(* Logix 5000 project; controller BoilerDemo vendor 1 type 14 code 164 rev 33.11; software revision 33.03 *)

TASK BoilerDemoTask (periodic, rate 75 ms, priority 10, watchdog 500 ms) : BoilerDemoProgram
TASK OvenDemoTask (continuous, watchdog 500 ms) : OvenDemo

MODULES
   Local : vendor 1 type 14 code 164 (ICP 1, rev 33.11)
END_MODULES

TYPE DATETIMESTRUCT :
STRUCT
   Year : DINT;
   Month : DINT;
   Day : DINT;
   Hour : DINT;
   Minute : DINT;
   Second : DINT;
   Microsecond : DINT;
END_STRUCT
END_TYPE

TYPE Motor :
STRUCT
   Power : REAL;
   Speed : INT;
   CmdOffOn : BOOL;
   SetSpeed : INT;
   Status : BOOL;
END_STRUCT
END_TYPE

TYPE Product :
STRUCT
   Product_id : INT;
   Product_name : STRING;
   Brand_id : INT;
   Category_id : INT;
   model_year : INT;
   list_price : REAL;
END_STRUCT
END_TYPE

TYPE Step :
STRUCT
   Num : INT;
   Time : TIMER;
   Step_Complete : BOOL;
   Prompt : BOOL;
   Prompt_Desc : STRING;
   Description : STRING;
END_STRUCT
END_TYPE

TYPE TankUDT :
STRUCT
   ValveInStatus : BOOL;
   ValveInCmd : BOOL;
   ValveOutStatus : BOOL;
   ValveOutCmd : BOOL;
   Level : REAL;
   SetPoint : REAL;
END_STRUCT
END_TYPE

ADD_ON_INSTRUCTION AOI_FaultGen   (* revision 1.2, vendor Rockwell Automation, ExecuteEnableInFalse *)
// Using random numbers [AOI_SIM_RNG_Simple] to generate 1-64 faults and their duration
// Revision note:
// Cfg_CycleTime changed to local tag (no need to have many configuration tags exposed)
// Help:
// This AOI uses Random Number ganerator to create up to 64 different outputus (BOOLs), each with different duration.
// ( Cfg_FaultOccurencesAll ) affects "probability" of TRUE value of all outputs ( F.x )
// ( Cfg_FaultOccurences[x] ) can be used to set the ratio among "probabilities" of individual outputs ( F.x ) getting true -> higher value, haigher probability
// Mechanism:
// - Value of the random number is between 0 and 1
// - Random number is generated every ( Cfg_CycleTime ) seconds
// - Value of Random numebr is checked, whether it falls in interval [0 - Cfg_FaultOccurenceAll]
// - If Random number is in the configured interval, then this interval is split into pieces:
//    where number of pieces to "split the interval into" is:
//    SUM of ( Cfg_FaultOccurences[] ) ... the count of Cfg_FaultOccurences members to use is ( Cfg_NumberOfFaults )
// - Each "output" (F.x) then has its "own" interval of the [0 - Cfg_FaultOccurenceAll]. If the Random number falls into the interval related to F.x, then F.x is set high
// - Reset of F.x to low is after a random time between ( Cfg_FaultDurationMin ) and ( Cfg_FaultDurationMax )
VAR_INPUT
   Cfg_NumberOfFaults : DINT := 1; {access None, visible}   // Number of faults to be generated (valid 1-64) value 0 resets the F (output) bits
   Cfg_FaultOccurenceAll : REAL := 0.05; {access None, visible}   // Probability of ANY fault occurence (valid 0-1)
   Cfg_FaultDurationMin : DINT := 15; {access None, visible}   // Minimum duration of fault [seconds]
   Cfg_FaultDurationMax : DINT := 75; {access None, visible}   // Maximum duration of fault [seconds]
END_VAR
VAR_OUTPUT
   F : LINT; {access None, visible}   // Generated fault bits
   RandomNr : REAL; {access Read Only, visible}
END_VAR
VAR
   TONs_FaultHold : TIMER[64]; {access None}
   z_CTRL : CONTROL := (LEN := 1); {access None}
   RandomNumber : REAL; {access None}
   TON_Cycle : TIMER := (PRE := 1500); {access None}
   Wrk_FaultOccurencesSUM : DINT; {access None}
   Wrk_Step : REAL; {access None}
   i : DINT; {access None}
   Wrk_StepLimit1 : REAL; {access None}
   Wrk_StepLimit2 : REAL; {access None}
   z_ONS : BOOL[64]; {access None}
   Random : AOI_SIM_RNG_Simple := (Seed := 521288629); {access None}
   Cfg_FaultOccurences : DINT[64] := ([0] := 100, [1] := 100, [2] := 100, [3] := 100, [4] := 100, [5] := 100, [6] := 100, [7] := 100, [8] := 100, [9] := 100, [10] := 100, [11] := 100, [12] := 100, [13] := 100, [14] := 100, [15] := 100, [16] := 100, [17] := 100, [18] := 100, [19] := 100, [20] := 100, [21] := 100, [22] := 100, [23] := 100, [24] := 100, [25] := 100, [26] := 100, [27] := 100, [28] := 100, [29] := 100, [30] := 100, [31] := 100, [32] := 100, [33] := 100, [34] := 100, [35] := 100, [36] := 100, [37] := 100, [38] := 100, [39] := 100, [40] := 100, [41] := 100, [42] := 100, [43] := 100, [44] := 100, [45] := 100, [46] := 100, [47] := 100, [48] := 100, [49] := 100, [50] := 100, [51] := 100, [52] := 100, [53] := 100, [54] := 100, [55] := 100, [56] := 100, [57] := 100, [58] := 100, [59] := 100,
        [60] := 100, [61] := 100, [62] := 100, [63] := 100);   // Each fault's "probability weight" (proportional to the other faults' "weights")
   i_max : DINT; {access None}
   Cfg_CycleTime : REAL := 1.5;   // Fault generation cycle time [seconds]
END_VAR

ROUTINE EnableInFalse   (* ladder *)
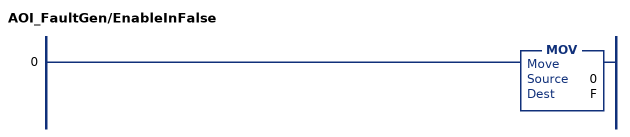
   0: MOV(0,F);
END_ROUTINE

ROUTINE Logic   (* ladder *)
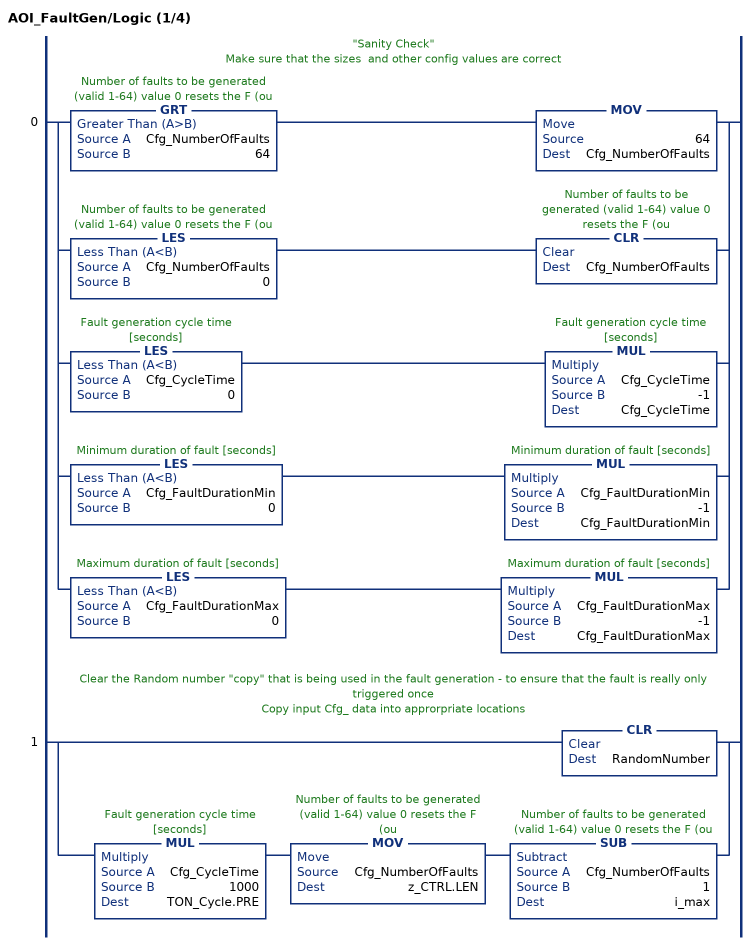
   // "Sanity Check"
   // Make sure that the sizes  and other config values are correct
   0: [GRT(Cfg_NumberOfFaults,64) MOV(64,Cfg_NumberOfFaults) ,LES(Cfg_NumberOfFaults,0) CLR(Cfg_NumberOfFaults) ,LES(Cfg_CycleTime,0) MUL(Cfg_CycleTime,-1,Cfg_CycleTime) ,LES(Cfg_FaultDurationMin,0) MUL(Cfg_FaultDurationMin,-1,Cfg_FaultDurationMin) ,LES(Cfg_FaultDurationMax,0) MUL(Cfg_FaultDurationMax,-1,Cfg_FaultDurationMax) ];
   // Clear the Random number "copy" that is being used in the fault generation - to ensure that the fault is really only triggered once
   // Copy input Cfg_ data into approrpriate locations
   1: [CLR(RandomNumber) ,MUL(Cfg_CycleTime,1000,TON_Cycle.PRE) MOV(Cfg_NumberOfFaults,z_CTRL.LEN) SUB(Cfg_NumberOfFaults,1,i_max) ];
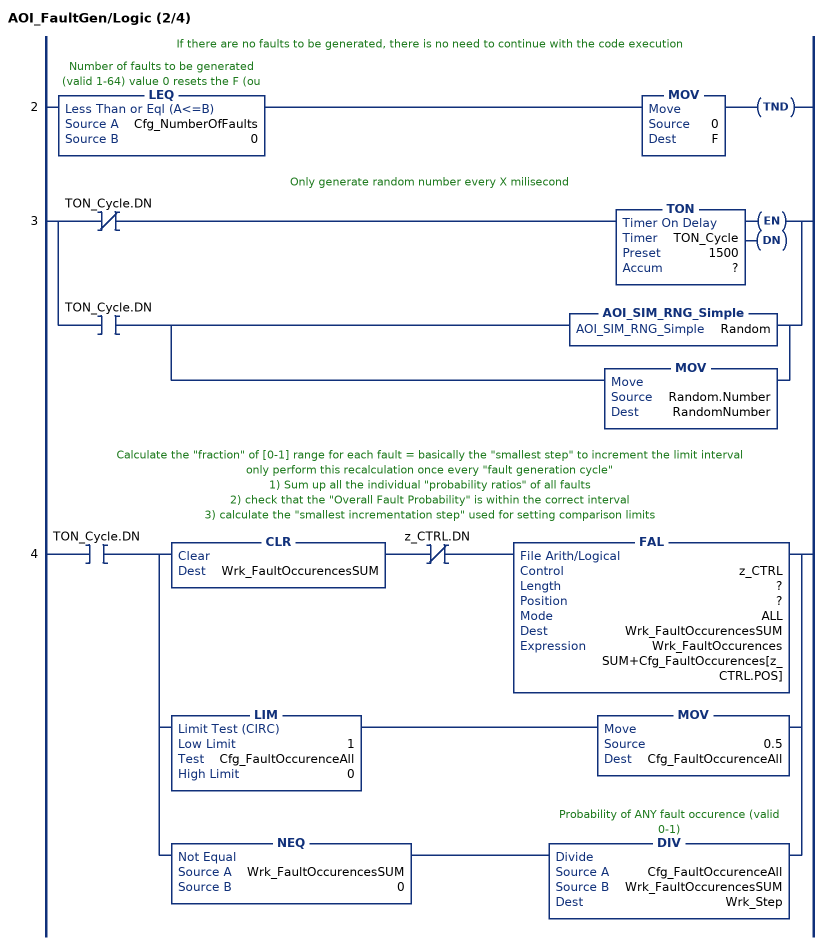
   // If there are no faults to be generated, there is no need to continue with the code execution
   2: LEQ(Cfg_NumberOfFaults,0)MOV(0,F)TND();
   // Only generate random number every X milisecond
   3: [XIO(TON_Cycle.DN) TON(TON_Cycle,?,?) ,XIC(TON_Cycle.DN) [AOI_SIM_RNG_Simple(Random) ,MOV(Random.Number,RandomNumber) ] ];
   // Calculate the "fraction" of [0-1] range for each fault = basically the "smallest step" to increment the limit interval
   // only perform this recalculation once every "fault generation cycle"
   // 1) Sum up all the individual "probability ratios" of all faults
   // 2) check that the "Overall Fault Probability" is within the correct interval
   // 3) calculate the "smallest incrementation step" used for setting comparison limits
   4: XIC(TON_Cycle.DN)[CLR(Wrk_FaultOccurencesSUM) XIO(z_CTRL.DN) FAL(z_CTRL,?,?,ALL,Wrk_FaultOccurencesSUM,Wrk_FaultOccurencesSUM+Cfg_FaultOccurences[z_CTRL.POS]) ,LIM(1,Cfg_FaultOccurenceAll,0) MOV(0.5,Cfg_FaultOccurenceAll) ,NEQ(Wrk_FaultOccurencesSUM,0) DIV(Cfg_FaultOccurenceAll,Wrk_FaultOccurencesSUM,Wrk_Step) ];
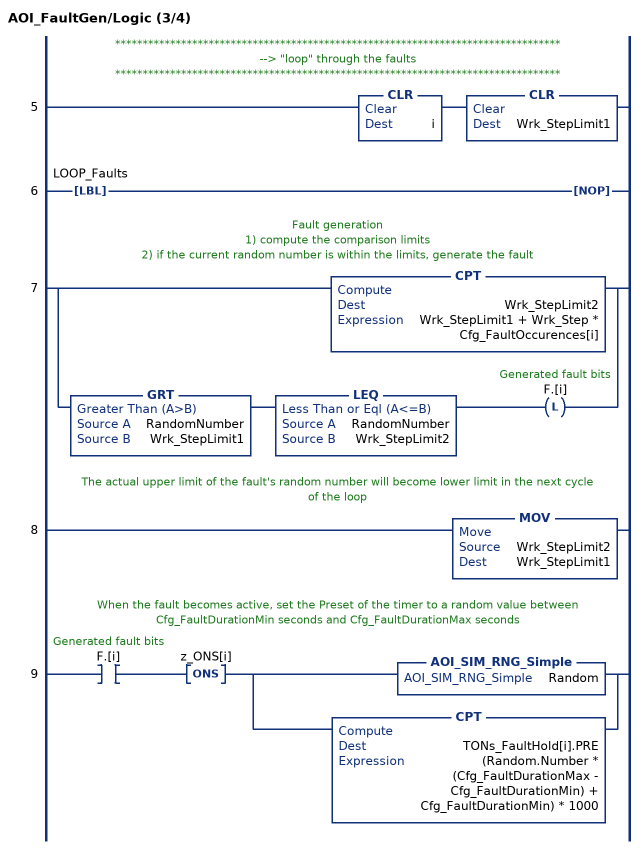
   // *********************************************************************************
   // --> "loop" through the faults
   // *********************************************************************************
   5: CLR(i)CLR(Wrk_StepLimit1);
   6: LBL(LOOP_Faults)NOP();
   // Fault generation
   // 1) compute the comparison limits
   // 2) if the current random number is within the limits, generate the fault
   7: [CPT(Wrk_StepLimit2,Wrk_StepLimit1 + Wrk_Step * Cfg_FaultOccurences[i]) ,GRT(RandomNumber,Wrk_StepLimit1) LEQ(RandomNumber,Wrk_StepLimit2) OTL(F.[i]) ];
   // The actual upper limit of the fault's random number will become lower limit in the next cycle of the loop
   8: MOV(Wrk_StepLimit2,Wrk_StepLimit1);
   // When the fault becomes active, set the Preset of the timer to a random value between Cfg_FaultDurationMin seconds and Cfg_FaultDurationMax seconds
   9: XIC(F.[i])ONS(z_ONS[i])[AOI_SIM_RNG_Simple(Random) ,CPT(TONs_FaultHold[i].PRE,(Random.Number * (Cfg_FaultDurationMax - Cfg_FaultDurationMin) + Cfg_FaultDurationMin) * 1000) ];
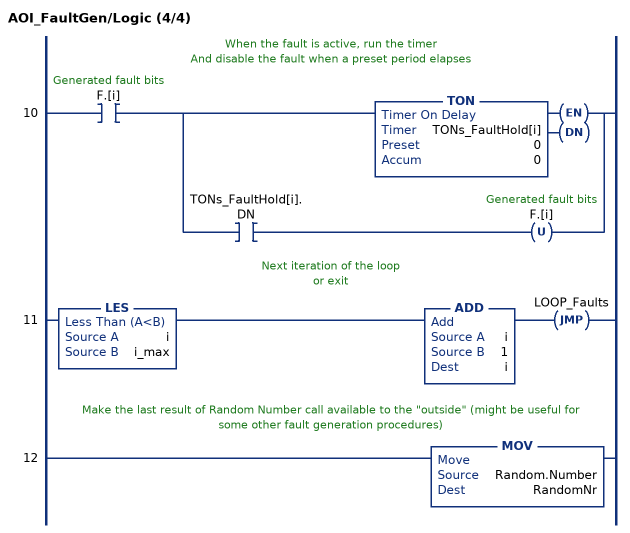
   // When the fault is active, run the timer
   // And disable the fault when a preset period elapses
   10: XIC(F.[i])[TON(TONs_FaultHold[i],0,0) ,XIC(TONs_FaultHold[i].DN) OTU(F.[i]) ];
   // Next iteration of the loop
   // or exit
   11: LES(i,i_max)ADD(i,1,i)JMP(LOOP_Faults);
   // Make the last result of Random Number call available to the "outside" (might be useful for some other fault generation procedures)
   12: MOV(Random.Number,RandomNr);
END_ROUTINE
END_ADD_ON_INSTRUCTION

ADD_ON_INSTRUCTION AOI_SIM_RNG_Simple   (* revision 1.3, vendor Dr. Frank Jordan / Rockwell Automation, ExecutePrescan *)
// Simple Random Number Generator
// Revision note:
// This code is provided as application example without any warranty
// Help:
// George Marsaglia 's MWC (multiply with carry) algorithm
// (taken from http://www.codeproject.com/Articles/25172/Simple-Random-Number-Generation)
VAR_INPUT
   Seed : ALIAS FOR LocalSeed; {access Read Only, visible}
END_VAR
VAR_OUTPUT
   Count : DINT; {access Read Only, visible}
   Number : REAL; {access Read Only, visible}
END_VAR
VAR_INPUT
   TriggerSeed : ALIAS FOR LocalTriggerSeed; {access Read Only, visible}
   Reset : ALIAS FOR LocalReset; {access Read Only, visible}
END_VAR
VAR
   m_z : DINT; {access None}
   m_w : DINT; {access None}
   delta : REAL; {access None}
   consB : DINT; {access None}
   consA : DINT; {access None}
   AOI_UMUL : UMUL; {access None}
   u : DINT; {access None}
   AOI_UADD : UADD; {access None}
   LocalTriggerSeed : BOOL; {access Read Only}
   LocalSeed : DINT; {access Read Only}
   LocalReset : BOOL; {access Read Only}
   tmp : DINT; {access None}
   Overflow : BOOL; {access None}
END_VAR

ROUTINE Logic   (* ladder *)
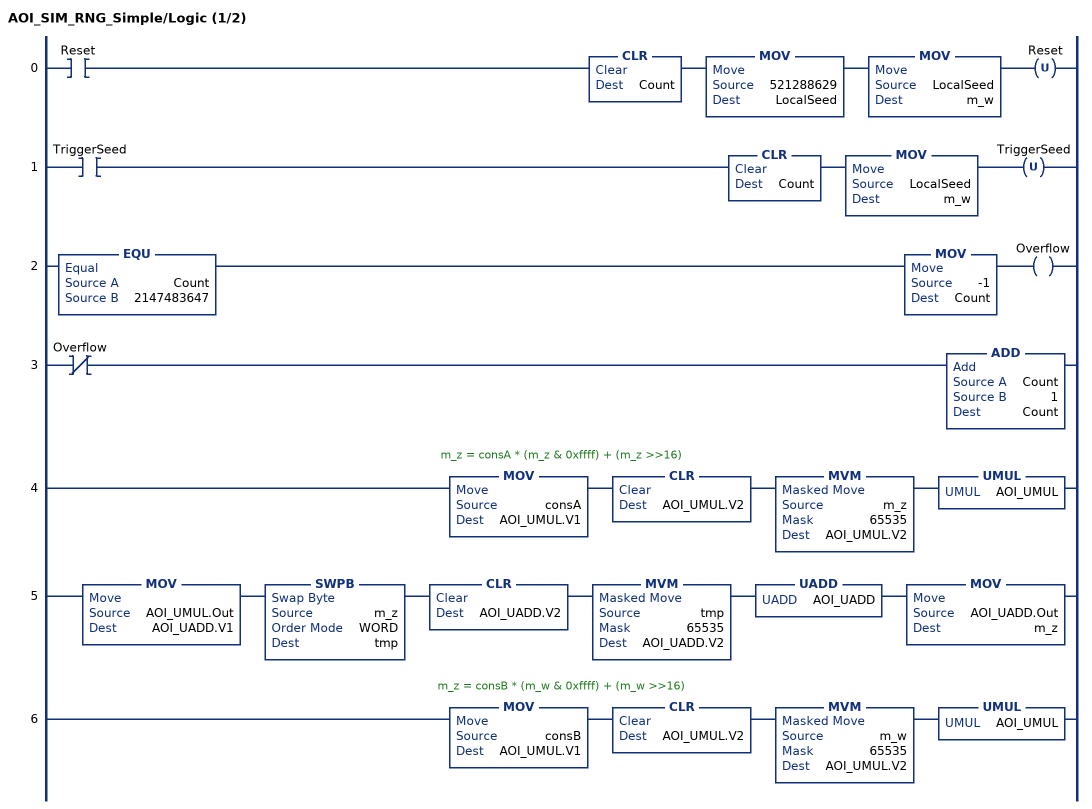
   0: XIC(Reset)CLR(Count)MOV(521288629,LocalSeed)MOV(LocalSeed,m_w)OTU(Reset);
   1: XIC(TriggerSeed)CLR(Count)MOV(LocalSeed,m_w)OTU(TriggerSeed);
   2: EQU(Count,2147483647)MOV(-1,Count)OTE(Overflow);
   3: XIO(Overflow)ADD(Count,1,Count);
   // m_z = consA * (m_z & 0xffff) + (m_z >>16)
   4: MOV(consA,AOI_UMUL.V1)CLR(AOI_UMUL.V2)MVM(m_z,65535,AOI_UMUL.V2)UMUL(AOI_UMUL);
   5: MOV(AOI_UMUL.Out,AOI_UADD.V1)SWPB(m_z,WORD,tmp)CLR(AOI_UADD.V2)MVM(tmp,65535,AOI_UADD.V2)UADD(AOI_UADD)MOV(AOI_UADD.Out,m_z);
   // m_z = consB * (m_w & 0xffff) + (m_w >>16)
   6: MOV(consB,AOI_UMUL.V1)CLR(AOI_UMUL.V2)MVM(m_w,65535,AOI_UMUL.V2)UMUL(AOI_UMUL);
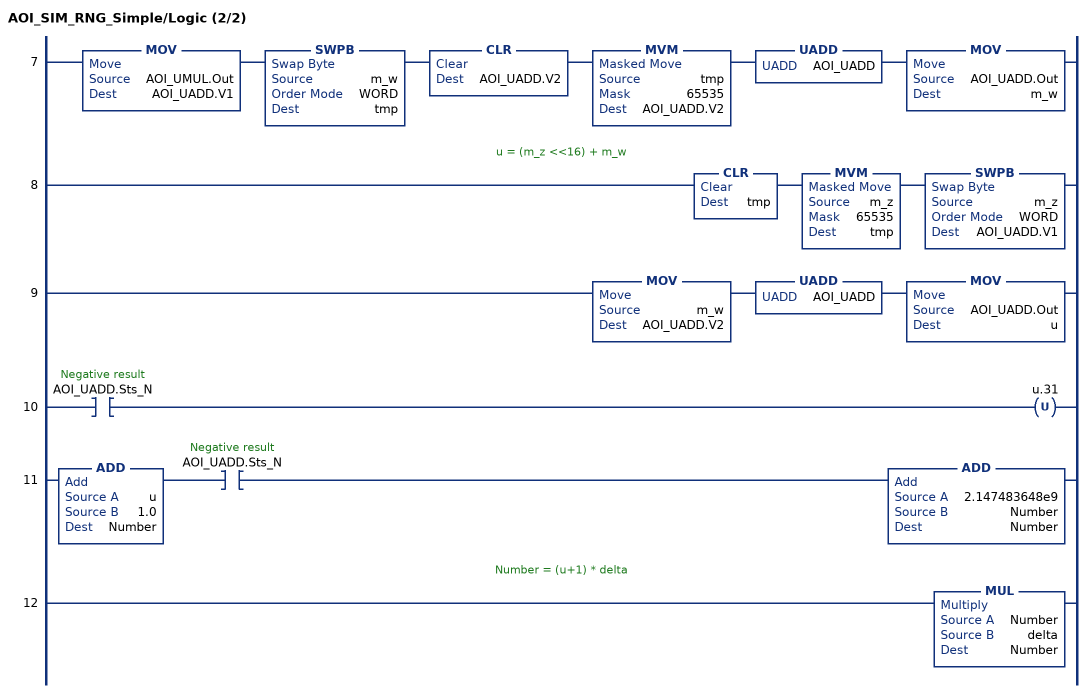
   7: MOV(AOI_UMUL.Out,AOI_UADD.V1)SWPB(m_w,WORD,tmp)CLR(AOI_UADD.V2)MVM(tmp,65535,AOI_UADD.V2)UADD(AOI_UADD)MOV(AOI_UADD.Out,m_w);
   // u = (m_z <<16) + m_w
   8: CLR(tmp)MVM(m_z,65535,tmp)SWPB(m_z,WORD,AOI_UADD.V1);
   9: MOV(m_w,AOI_UADD.V2)UADD(AOI_UADD)MOV(AOI_UADD.Out,u);
   10: XIC(AOI_UADD.Sts_N)OTU(u.31);
   11: ADD(u,1.0,Number)XIC(AOI_UADD.Sts_N)ADD(2.147483648e9,Number,Number);
   // Number = (u+1) * delta
   12: MUL(Number,delta,Number);
END_ROUTINE

ROUTINE Prescan   (* ladder *)
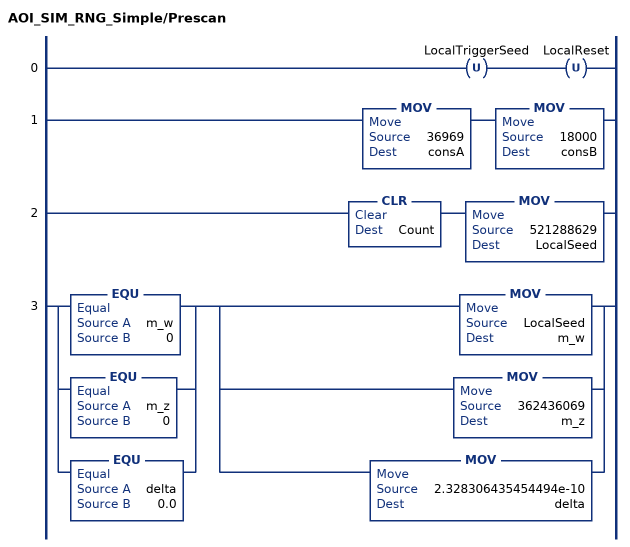
   0: OTU(LocalTriggerSeed)OTU(LocalReset);
   1: MOV(36969,consA)MOV(18000,consB);
   2: CLR(Count)MOV(521288629,LocalSeed);
   3: [EQU(m_w,0) ,EQU(m_z,0) ,EQU(delta,0.0) ][MOV(LocalSeed,m_w) ,MOV(362436069,m_z) ,MOV(2.328306435454494e-10,delta) ];
END_ROUTINE
END_ADD_ON_INSTRUCTION

ADD_ON_INSTRUCTION UADD   (* revision 1.1, vendor Dr. Frank Jordan / Rockwell Automation *)
// Addition of  two unsigned DINT
// (without overflow / minor faults)
// Revision note:
// This code is provided as application example without any warranty
VAR_INPUT
   V1 : DINT; {visible}
   V2 : DINT; {visible}
END_VAR
VAR_OUTPUT
   Out : DINT; {access Read Only, visible}
   Sts_C : BOOL; {access Read Only, visible}   // Carry result
   Sts_N : BOOL; {access Read Only, visible}   // Negative result
   Sts_V : BOOL; {access Read Only, visible}   // Overflow result
   Sts_Z : BOOL; {access Read Only, visible}   // Zero result
END_VAR
VAR
   V1_Hi : DINT; {access None}
   V1_Lo : DINT; {access None}
   V2_Hi : DINT; {access None}
   V2_Lo : DINT; {access None}
   SumLo : DINT; {access None}
   SumHi : DINT; {access None}
   tmp : DINT; {access None}
END_VAR

ROUTINE Logic   (* ladder *)
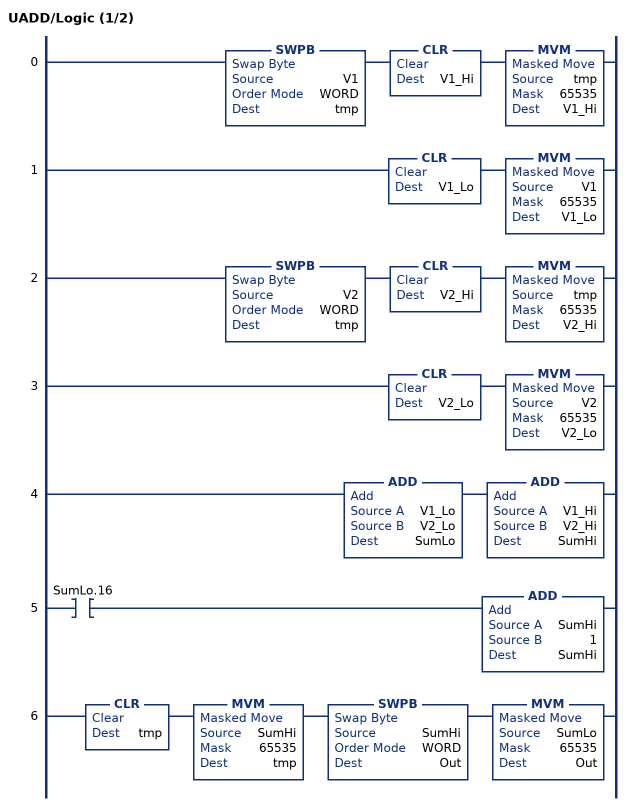
   0: SWPB(V1,WORD,tmp)CLR(V1_Hi)MVM(tmp,65535,V1_Hi);
   1: CLR(V1_Lo)MVM(V1,65535,V1_Lo);
   2: SWPB(V2,WORD,tmp)CLR(V2_Hi)MVM(tmp,65535,V2_Hi);
   3: CLR(V2_Lo)MVM(V2,65535,V2_Lo);
   4: ADD(V1_Lo,V2_Lo,SumLo)ADD(V1_Hi,V2_Hi,SumHi);
   5: XIC(SumLo.16)ADD(SumHi,1,SumHi);
   6: CLR(tmp)MVM(SumHi,65535,tmp)SWPB(SumHi,WORD,Out)MVM(SumLo,65535,Out);
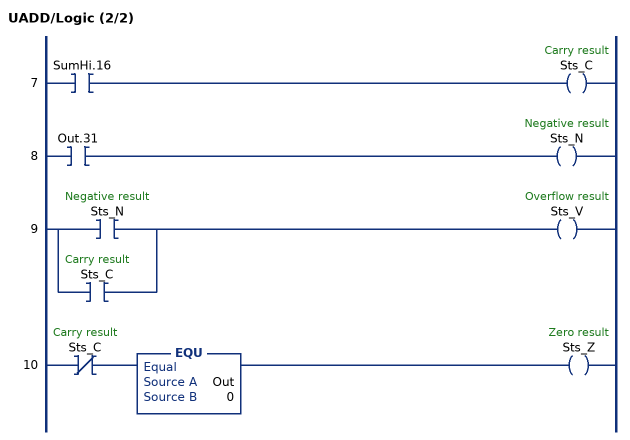
   7: XIC(SumHi.16)OTE(Sts_C);
   8: XIC(Out.31)OTE(Sts_N);
   9: [XIC(Sts_N) ,XIC(Sts_C) ]OTE(Sts_V);
   10: XIO(Sts_C)EQU(Out,0)OTE(Sts_Z);
END_ROUTINE
END_ADD_ON_INSTRUCTION

ADD_ON_INSTRUCTION UMUL   (* revision 1.2, vendor Dr. Frank Jordan / Rockwell Automation *)
// Multiplication of  two unsigned DINT
// (without overflow / minor faults)
// Revision note:
// This code is provided as application example without any warranty
VAR_INPUT
   V1 : DINT; {visible}
   V2 : DINT; {visible}
END_VAR
VAR_OUTPUT
   Sts_C : BOOL; {access Read Only, visible}   // Carry result
   Sts_N : BOOL; {access Read Only, visible}   // Negative result
   Sts_V : BOOL; {access Read Only, visible}   // Overflow result
   Sts_Z : BOOL; {access Read Only, visible}   // Zero result
   Out : DINT; {access Read Only, visible}
END_VAR
VAR
   tmp : DINT; {access None}
   WRK : INT[6]; {access None}
   WRKm : DINT[6]; {access None}
   Low : DINT; {access None}
   Mid : DINT; {access None}
   High : DINT; {access None}
END_VAR

ROUTINE Logic   (* ladder *)
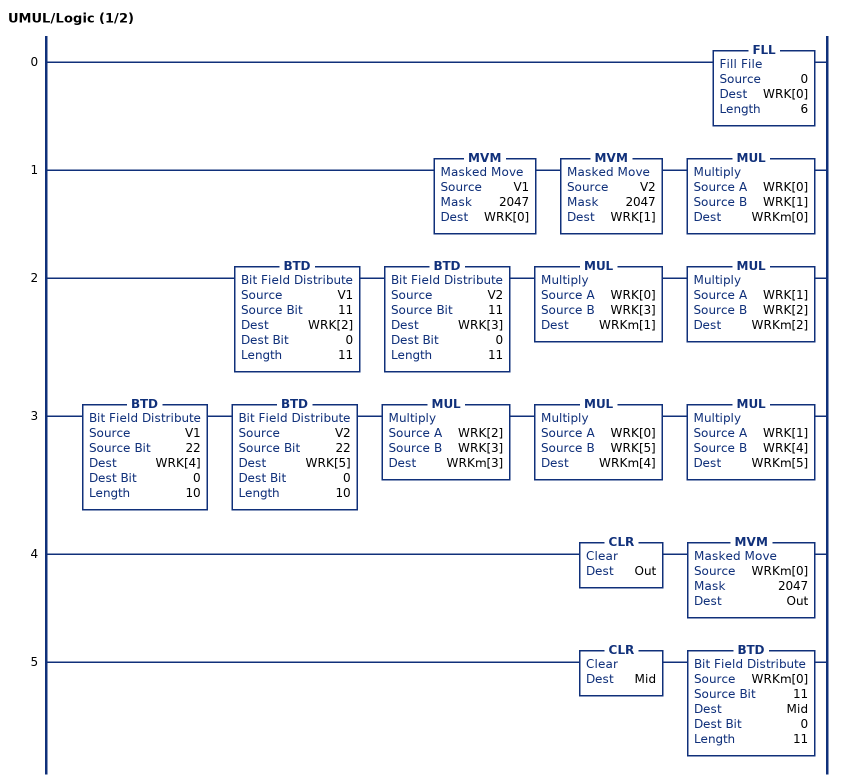
   0: FLL(0,WRK[0],6);
   1: MVM(V1,2047,WRK[0])MVM(V2,2047,WRK[1])MUL(WRK[0],WRK[1],WRKm[0]);
   2: BTD(V1,11,WRK[2],0,11)BTD(V2,11,WRK[3],0,11)MUL(WRK[0],WRK[3],WRKm[1])MUL(WRK[1],WRK[2],WRKm[2]);
   3: BTD(V1,22,WRK[4],0,10)BTD(V2,22,WRK[5],0,10)MUL(WRK[2],WRK[3],WRKm[3])MUL(WRK[0],WRK[5],WRKm[4])MUL(WRK[1],WRK[4],WRKm[5]);
   4: CLR(Out)MVM(WRKm[0],2047,Out);
   5: CLR(Mid)BTD(WRKm[0],11,Mid,0,11);
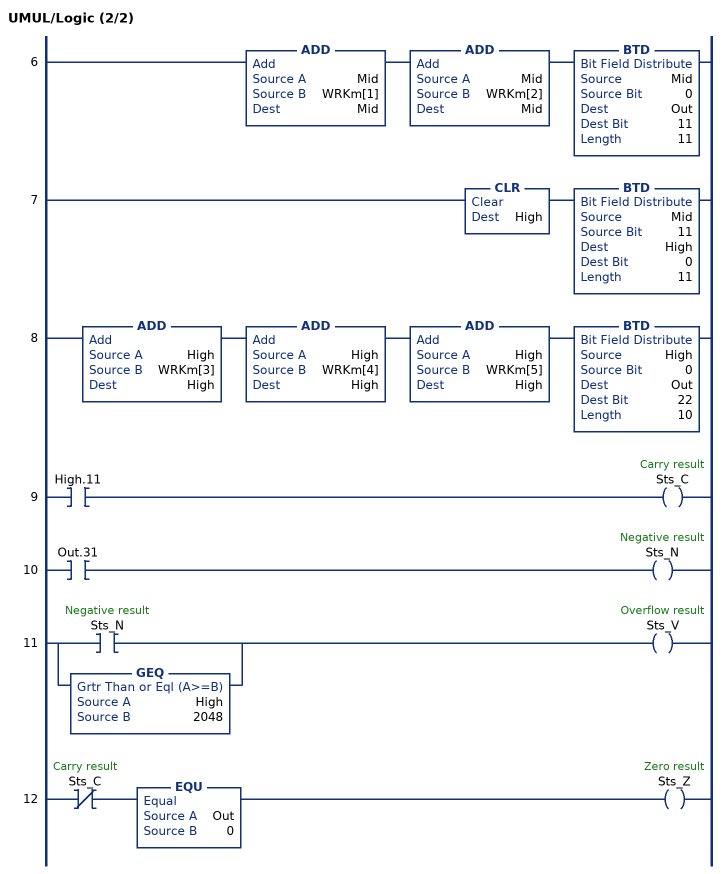
   6: ADD(Mid,WRKm[1],Mid)ADD(Mid,WRKm[2],Mid)BTD(Mid,0,Out,11,11);
   7: CLR(High)BTD(Mid,11,High,0,11);
   8: ADD(High,WRKm[3],High)ADD(High,WRKm[4],High)ADD(High,WRKm[5],High)BTD(High,0,Out,22,10);
   9: XIC(High.11)OTE(Sts_C);
   10: XIC(Out.31)OTE(Sts_N);
   11: [XIC(Sts_N) ,GEQ(High,2048) ]OTE(Sts_V);
   12: XIO(Sts_C)EQU(Out,0)OTE(Sts_Z);
END_ROUTINE
END_ADD_ON_INSTRUCTION

VAR_GLOBAL   (* controller tags *)
   Motors : Motor[5] := ([0].Power := -0.2, [0].Speed := -1, [0].SetSpeed := 100, [1].Power := -0.2, [1].Speed := -1, [1].SetSpeed := 120, [2].Power := -0.2, [2].Speed := -1, [2].SetSpeed := 140, [3].Power := -0.2, [3].Speed := -1, [3].SetSpeed := 160, [4].Power := -0.2, [4].Speed := -1, [4].SetSpeed := 180);
   Product_Selected_Bike : Product := (Product_id := 102, Product_name := 'Electra Townie Original 7D - 2017', Brand_id := 1, Category_id := 2, model_year := 2017, list_price := 489.99);
   Pump : Motor[20] := ([0].Power := 12.0, [0].Speed := 22, [0].SetSpeed := 13, [1].Speed := 55, [1].SetSpeed := 56, [1].Status := 1, [2].Speed := 33);
   Tank1 : TankUDT := (ValveInCmd := 1, Level := 49.0, SetPoint := 50.0);
   Tank2 : TankUDT := (ValveInCmd := 1, Level := 49.0, SetPoint := 50.0);
   TestBoolTag : BOOL;
   TestIncrementTag : DINT;
END_VAR

PROGRAM BoilerDemoProgram   (* main routine BoilerDemoRoutine *)
VAR
   Count : INT := 5;
   Direction : BOOL := 1;
   Init : BOOL := 1;
END_VAR

ROUTINE BoilerDemoRoutine   (* structured text *)
   //Init Motors and WaterTank
   if (not Init) then
   	Init := 1;
   	Motors[0].SetSpeed := 100;
   	Motors[1].SetSpeed := 120;
   	Motors[2].SetSpeed := 140;
   	Motors[3].SetSpeed := 160;
   	Motors[4].SetSpeed := 180;
   	Tank2.SetPoint := 50.0;
   	Tank1.SetPoint := 50.0;
   	Tank2.Level := 1;
   	Tank1.Level := 1;
   end_if;
   
   if (TestIncrementTag = 0) then
   	Direction := 1;
   end_if;
   if (TestIncrementTag = 100) then
   	Direction := 0;
   end_if;
   if (TestBoolTag) then
   	if (Direction) then
   		TestIncrementTag := TestIncrementTag + 1;
   	else
   		TestIncrementTag := TestIncrementTag - 1;
   	end_if;
   end_if;
   
   //Tank 2 Logic
   if (Tank2.ValveInCmd) then
   	if (Tank2.Level < (Tank2.SetPoint - 1)) then
   		Tank2.ValveInStatus := 1;
   		Tank2.Level := Tank2.Level + 1;
   	else
   		Tank2.ValveInStatus := 0;
   	end_if;
   else
   	Tank2.ValveInStatus := 0;
   end_if;
   
   if (Tank2.ValveOutCmd) then
   	if (Tank2.Level >= 1)  then
   		Tank2.ValveOutStatus := 1;
   		Tank2.Level := Tank2.Level - 1;
   	else
   		Tank2.ValveOutStatus := 0;
   	end_if;
   else
   	Tank2.ValveOutStatus := 0;
   end_if;
   
   //Tank 1 Logic
   if (Tank1.ValveInCmd) then
   	if (Tank1.Level < (Tank1.SetPoint - 1)) then
   		Tank1.ValveInStatus := 1;
   		Tank1.Level := Tank1.Level + 1;
   	else
   		Tank1.ValveInStatus := 0;
   	end_if;
   else
   	Tank1.ValveInStatus := 0;
   end_if;
   
   if (Tank1.ValveOutCmd) then
   	if (Tank1.Level >= 1) then
   		Tank1.ValveOutStatus := 1;
   		Tank1.Level := Tank1.Level - 1;
   	else
   		Tank1.ValveOutStatus := 0;
   	end_if;
   else
   	Tank1.ValveOutStatus := 0;
   end_if;
   
   //Motor Logic
   for Count := 0 to 4 do
   	if (Motors[Count].CmdOffOn) then
   		Motors[Count].Status := 1;
   		if (Motors[Count].Speed <= Motors[Count].SetSpeed) then
   			Motors[Count].Speed := Motors[Count].Speed + 1;
   			Motors[Count].Power := Motors[Count].Power + 0.2;
   		end_if;
   	else
   		Motors[Count].Status := 0;
   		if (Motors[Count].Speed >= 0) then
   			Motors[Count].Speed := Motors[Count].Speed - 1;
   			Motors[Count].Power := Motors[Count].Power - 0.2;
   		end_if;
   	end_if;
   end_for;
   
END_ROUTINE
END_PROGRAM

PROGRAM OvenDemo   (* main routine MainRoutine *)
VAR
   ActualDuration : DINT := 71; {access Read Only}
   ActualDuration_F : DINT[4] := ([1] := 15, [2] := 30, [3] := 25); {access Read Only}   // Actual Duration (Phases)
        [0]   // DO NOT USE
   ActualPhase : DINT; {access Read Only}
   ActualSetpoint : DINT := 120; {access Read Only}   // Actual temperature setpoint (for current phase)
   ActualTemperature : REAL := 1.1170044e-37; {access Read Only}
   Count : INT;
   CycleNumber : DINT := 33;
   Direction : BOOL;
   DoorAlarm : BOOL; {access Read Only}
   FanAlarm : BOOL; {access Read Only}
   FilterAlarm : BOOL; {access Read Only}
   Gas : REAL := 0.0056216787; {access Read Only}
   GasThrottle : REAL; {access Read Only}
   Init : BOOL;
   JobFinish : DATETIMESTRUCT := (Year := 1998, Month := 3, Day := 8, Hour := 23, Minute := 47, Second := 56, Microsecond := 247241); {access Read Only}
   JobGas : REAL := 0.0056216787; {access Read Only}
   JobkWh : REAL := 0.045102727; {access Read Only}
   JobRecipe : STRING; {access Read Only}
   JobStart : DATETIMESTRUCT := (Year := 1998, Month := 3, Day := 8, Hour := 23, Minute := 46, Second := 46, Microsecond := 16656); {access Read Only}
   kW : REAL := 3.0; {access Read Only}
   kWh : REAL := 0.045102727; {access Read Only}
   Preheating : BOOL;
   RecipeName : STRING;   // Setpoint: Recipe Name
   ResetFilter : BOOL;   // Comand to reset filter
   Running : BOOL; {access Read Only}   // Status: Sequence is Running
   SET_Duration_F : DINT[4] := ([1] := 15, [2] := 30, [3] := 25);   // Setpoints: Duratino of phases
        [0]   // DO NOT USE
   SET_FilterLimit : DINT := 500;   // Setpoint: Filter Lifetime
   SET_PreheatingTemperature : DINT;   // Setpoint: Preheating Temperature
   SET_SpeedFanInput_F : DINT[4] := ([1] := 10, [2] := 20, [3] := 50);   // Setpoints: Fan Speed on Input
        [0]   // DO NOT USE
   SET_SpeedFanOutput_F : DINT[4] := ([1] := 15, [2] := 15, [3] := 50);   // Setpoints: Fan Speeds on Output
        [0]   // DO NOT USE
   SET_TemperatureSetpoint_F : DINT[4] := ([1] := 250, [2] := 270, [3] := 120);   // Setpoints: Temperatures in different phases
        [0]   // DO NOT USE
   SpeedFanInput : DINT; {access Read Only}   // Actual Speed: Input Fan
   SpeedFanOutput : DINT; {access Read Only}   // Actual Speed: Output Fan
   StartStop : BOOL;
   TemperatureAlarm : BOOL; {access Read Only}
   TimeToFinishAll : DINT := -1; {access Read Only}
   TimeToFinishPhase : DINT; {access Read Only}
   TotEE : REAL := 0.5501849;
   TotLPG : REAL := 0.19104695;
   UseMinute : DINT := 500; {access Read Only}
   WRK_Gas_change : REAL; {access None}
   WRK_interval : DINT := 24; {access None}   // Interval between scans (seconds)
   WRK_interval_CSTactual : DINT[2] := ([0] := 190188671, [1] := 2); {access None}
   WRK_interval_CSTprevious : DINT[2] := ([0] := 190188671); {access None}
   WRK_kWh_change : REAL := 0.00020833334; {access None}
   WRK_TemperatureSetpoint : REAL; {access None}
   WRK_throttle : REAL; {access None}
   WRK_TimeToFinishAll : REAL := -1.0461318; {access None}
   WRK_TimeToFinishPhase : REAL := -1.2949209e-05; {access None}
   WRK_useMinute : REAL := 499500000.0; {access None}
   zCTRL_Alarms : AOI_FaultGen := (Cfg_NumberOfFaults := 3, Cfg_FaultOccurenceAll := 0.05, Cfg_FaultDurationMin := 1, Cfg_FaultDurationMax := 5, RandomNr := 0.9478334); {access None}
        .F.2   // Door Alarm
        .F.1   // Fan Alarm
        .F.0   // Temperature Alarm
   zCTRL_Finished_STOP : BOOL; {access None}   // All phases finished, stop the sequence
   zCTRL_FirstRunBit : BOOL; {access None}   // First run after START command
   zCTRL_SetPointPhase : BOOL; {access None}   // Switch between phases
   zCTRL_Timer : TIMER := (PRE := 250, ACC := 159, EN := 1, TT := 1); {access None}
END_VAR

ROUTINE Alarms   (* ladder *)
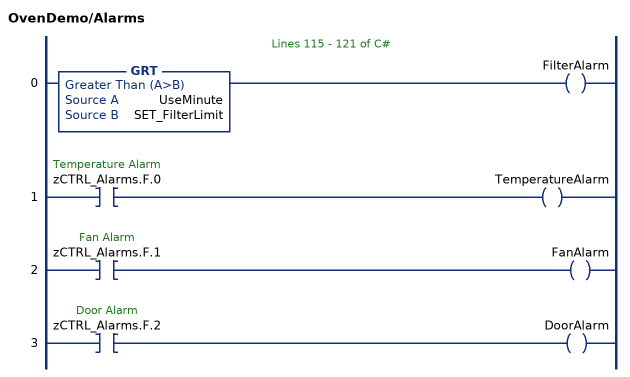
   // Lines 115 - 121 of C#
   0: GRT(UseMinute,SET_FilterLimit)OTE(FilterAlarm);
   1: XIC(zCTRL_Alarms.F.0)OTE(TemperatureAlarm);
   2: XIC(zCTRL_Alarms.F.1)OTE(FanAlarm);
   3: XIC(zCTRL_Alarms.F.2)OTE(DoorAlarm);
END_ROUTINE

ROUTINE MainRoutine   (* ladder *)
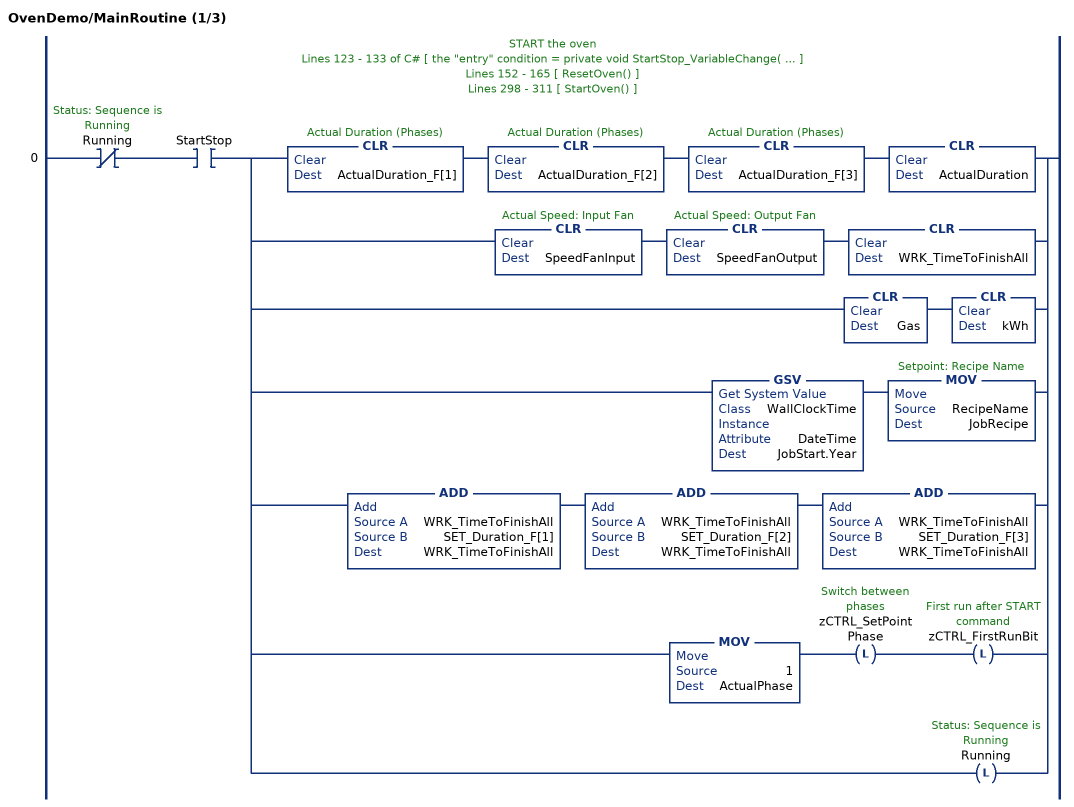
   // START the oven
   // Lines 123 - 133 of C# [ the "entry" condition = private void StartStop_VariableChange( ... ]
   // Lines 152 - 165 [ ResetOven() ]
   // Lines 298 - 311 [ StartOven() ]
   0: XIO(Running)XIC(StartStop)[CLR(ActualDuration_F[1]) CLR(ActualDuration_F[2]) CLR(ActualDuration_F[3]) CLR(ActualDuration) ,CLR(SpeedFanInput) CLR(SpeedFanOutput) CLR(WRK_TimeToFinishAll) ,CLR(Gas) CLR(kWh) ,GSV(WallClockTime,,DateTime,JobStart.Year) MOV(RecipeName,JobRecipe) ,ADD(WRK_TimeToFinishAll,SET_Duration_F[1],WRK_TimeToFinishAll) ADD(WRK_TimeToFinishAll,SET_Duration_F[2],WRK_TimeToFinishAll) ADD(WRK_TimeToFinishAll,SET_Duration_F[3],WRK_TimeToFinishAll) ,MOV(1,ActualPhase) OTL(zCTRL_SetPointPhase) OTL(zCTRL_FirstRunBit) ,OTL(Running) ];
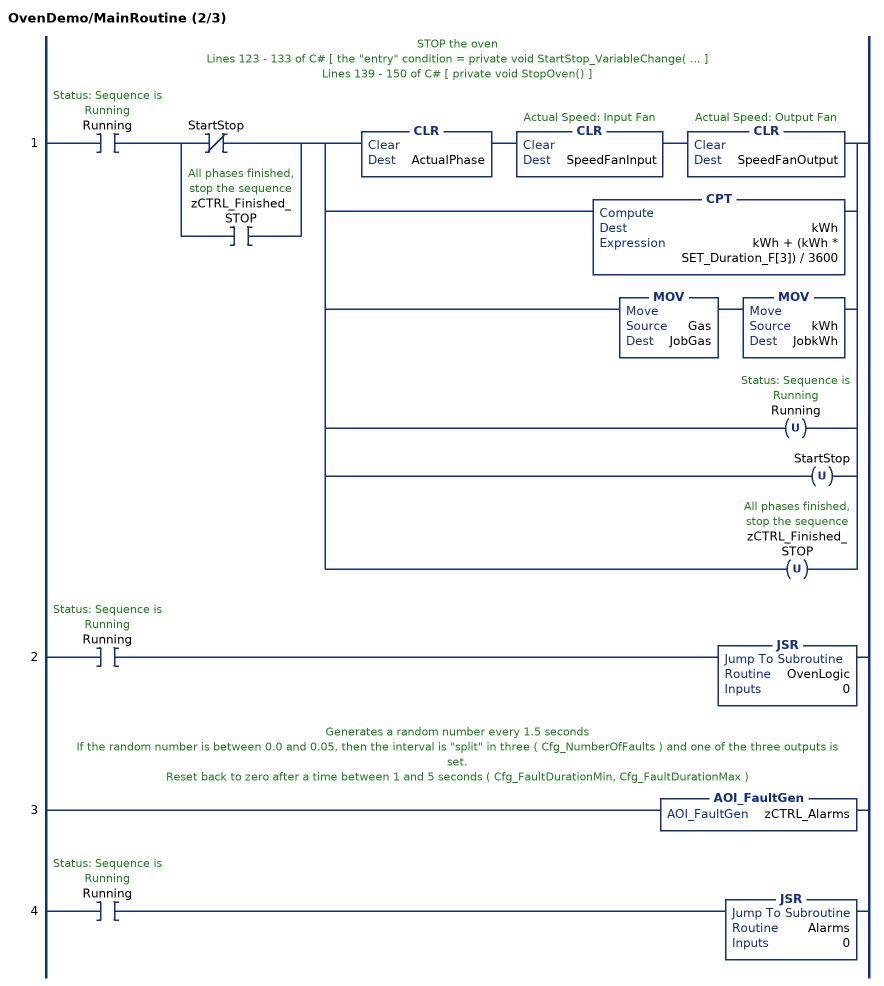
   // STOP the oven
   // Lines 123 - 133 of C# [ the "entry" condition = private void StartStop_VariableChange( ... ]
   // Lines 139 - 150 of C# [ private void StopOven() ]
   1: XIC(Running)[XIO(StartStop) ,XIC(zCTRL_Finished_STOP) ][CLR(ActualPhase) CLR(SpeedFanInput) CLR(SpeedFanOutput) ,CPT(kWh,kWh + (kWh * SET_Duration_F[3]) / 3600) ,MOV(Gas,JobGas) MOV(kWh,JobkWh) ,OTU(Running) ,OTU(StartStop) ,OTU(zCTRL_Finished_STOP) ];
   2: XIC(Running)JSR(OvenLogic,0);
   // Generates a random number every 1.5 seconds
   // If the random number is between 0.0 and 0.05, then the interval is "split" in three ( Cfg_NumberOfFaults ) and one of the three outputs is set.
   // Reset back to zero after a time between 1 and 5 seconds ( Cfg_FaultDurationMin, Cfg_FaultDurationMax )
   3: AOI_FaultGen(zCTRL_Alarms);
   4: XIC(Running)JSR(Alarms,0);
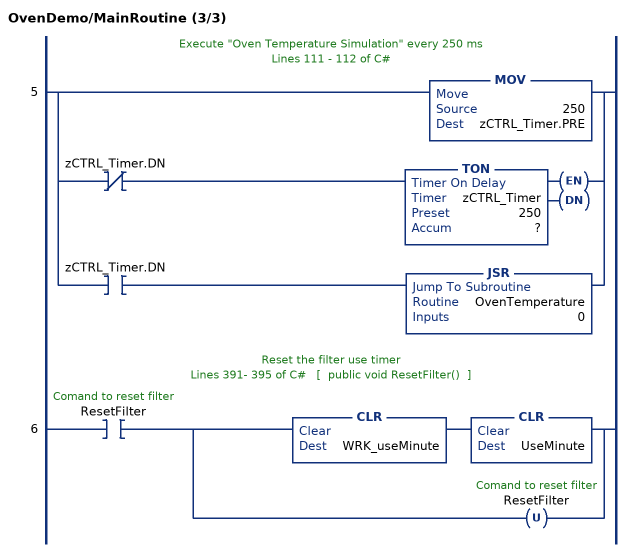
   // Execute "Oven Temperature Simulation" every 250 ms
   // Lines 111 - 112 of C#
   5: [MOV(250,zCTRL_Timer.PRE) ,XIO(zCTRL_Timer.DN) TON(zCTRL_Timer,?,?) ,XIC(zCTRL_Timer.DN) JSR(OvenTemperature,0) ];
   // Reset the filter use timer
   // Lines 391- 395 of C#   [  public void ResetFilter()  ]
   6: XIC(ResetFilter)[CLR(WRK_useMinute) CLR(UseMinute) ,OTU(ResetFilter) ];
END_ROUTINE

ROUTINE OvenLogic   (* ladder *)
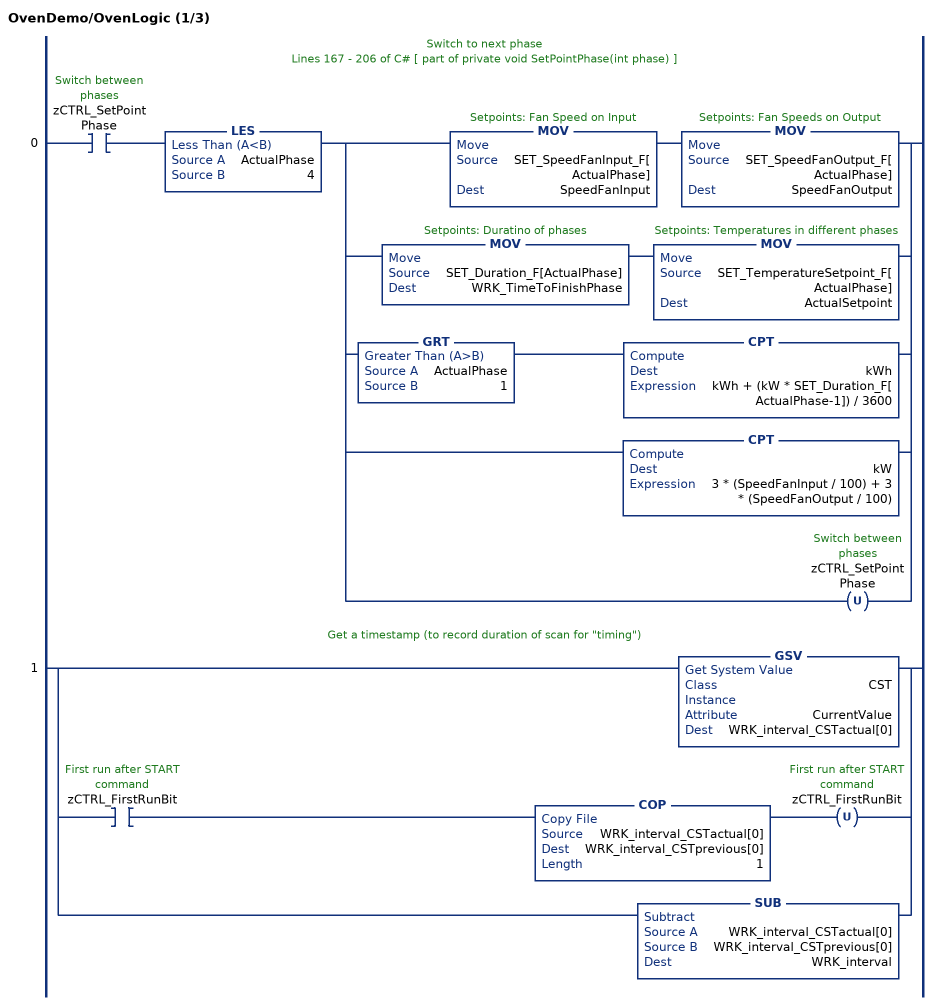
   // Switch to next phase
   // Lines 167 - 206 of C# [ part of private void SetPointPhase(int phase) ]
   0: XIC(zCTRL_SetPointPhase)LES(ActualPhase,4)[MOV(SET_SpeedFanInput_F[ActualPhase],SpeedFanInput) MOV(SET_SpeedFanOutput_F[ActualPhase],SpeedFanOutput) ,MOV(SET_Duration_F[ActualPhase],WRK_TimeToFinishPhase) MOV(SET_TemperatureSetpoint_F[ActualPhase],ActualSetpoint) ,GRT(ActualPhase,1) CPT(kWh,kWh + (kW * SET_Duration_F[ActualPhase-1]) / 3600) ,CPT(kW,3 * (SpeedFanInput / 100) + 3 * (SpeedFanOutput / 100)) ,OTU(zCTRL_SetPointPhase) ];
   // Get a timestamp (to record duration of scan for "timing")
   1: [GSV(CST,,CurrentValue,WRK_interval_CSTactual[0]) ,XIC(zCTRL_FirstRunBit) COP(WRK_interval_CSTactual[0],WRK_interval_CSTprevious[0],1) OTU(zCTRL_FirstRunBit) ,SUB(WRK_interval_CSTactual[0],WRK_interval_CSTprevious[0],WRK_interval) ];
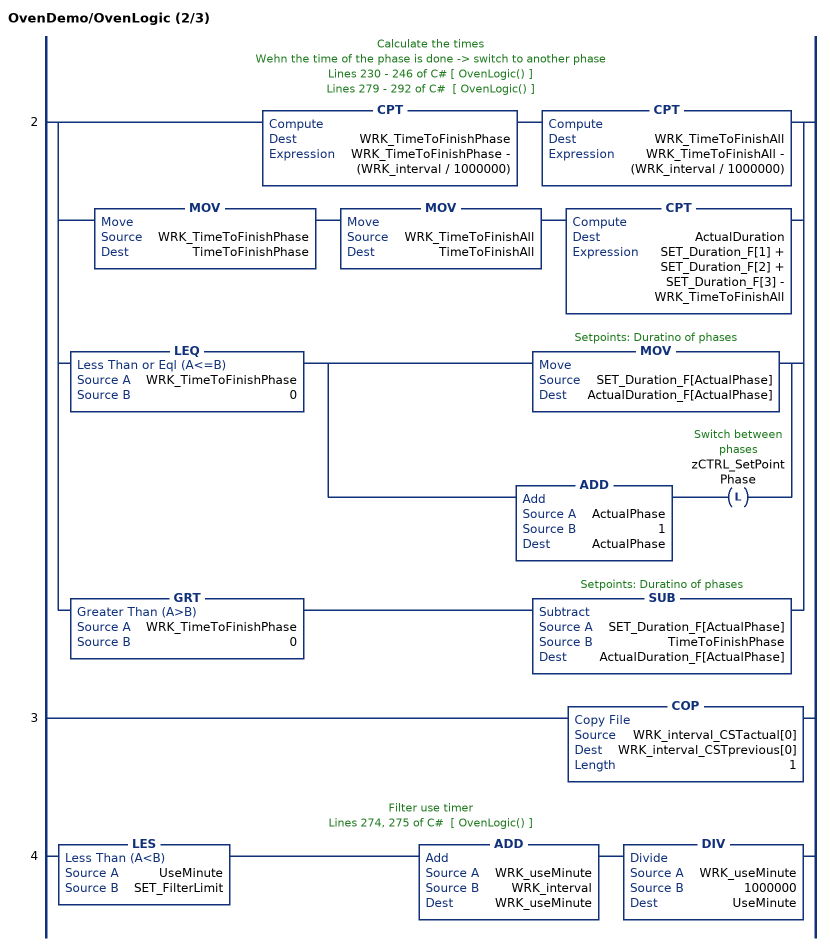
   // Calculate the times
   // Wehn the time of the phase is done -> switch to another phase
   // Lines 230 - 246 of C# [ OvenLogic() ]
   // Lines 279 - 292 of C#  [ OvenLogic() ]
   2: [[CPT(WRK_TimeToFinishPhase,WRK_TimeToFinishPhase - (WRK_interval / 1000000)) CPT(WRK_TimeToFinishAll,WRK_TimeToFinishAll - (WRK_interval / 1000000)) ,MOV(WRK_TimeToFinishPhase,TimeToFinishPhase) MOV(WRK_TimeToFinishAll,TimeToFinishAll) CPT(ActualDuration,SET_Duration_F[1] + SET_Duration_F[2] + SET_Duration_F[3] - WRK_TimeToFinishAll) ] ,LEQ(WRK_TimeToFinishPhase,0) [MOV(SET_Duration_F[ActualPhase],ActualDuration_F[ActualPhase]) ,ADD(ActualPhase,1,ActualPhase) OTL(zCTRL_SetPointPhase) ] ,GRT(WRK_TimeToFinishPhase,0) SUB(SET_Duration_F[ActualPhase],TimeToFinishPhase,ActualDuration_F[ActualPhase]) ];
   3: COP(WRK_interval_CSTactual[0],WRK_interval_CSTprevious[0],1);
   // Filter use timer
   // Lines 274, 275 of C#  [ OvenLogic() ]
   4: LES(UseMinute,SET_FilterLimit)ADD(WRK_useMinute,WRK_interval,WRK_useMinute)DIV(WRK_useMinute,1000000,UseMinute);
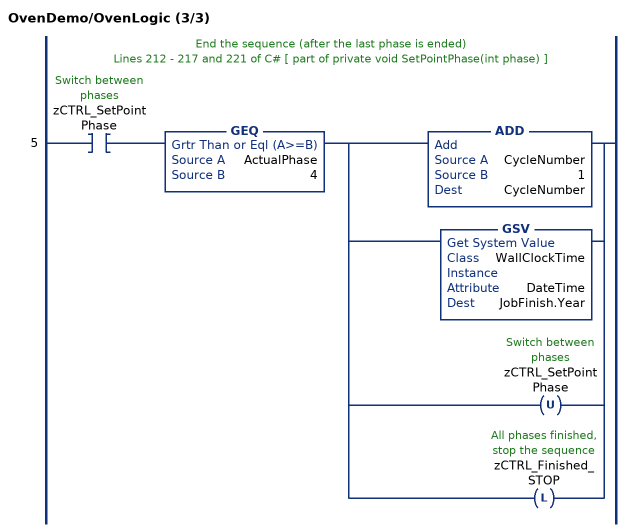
   // End the sequence (after the last phase is ended)
   // Lines 212 - 217 and 221 of C# [ part of private void SetPointPhase(int phase) ]
   5: XIC(zCTRL_SetPointPhase)GEQ(ActualPhase,4)[ADD(CycleNumber,1,CycleNumber) ,GSV(WallClockTime,,DateTime,JobFinish.Year) ,OTU(zCTRL_SetPointPhase) ,OTL(zCTRL_Finished_STOP) ];
END_ROUTINE

ROUTINE OvenTemperature   (* ladder *)
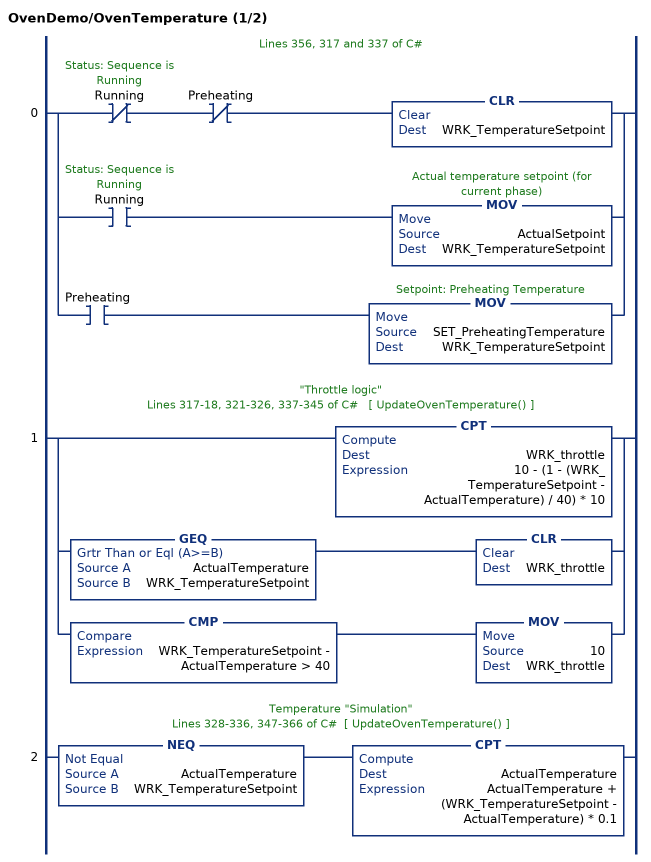
   // Lines 356, 317 and 337 of C#
   0: [XIO(Running) XIO(Preheating) CLR(WRK_TemperatureSetpoint) ,XIC(Running) MOV(ActualSetpoint,WRK_TemperatureSetpoint) ,XIC(Preheating) MOV(SET_PreheatingTemperature,WRK_TemperatureSetpoint) ];
   // "Throttle logic"
   // Lines 317-18, 321-326, 337-345 of C#   [ UpdateOvenTemperature() ]
   1: [CPT(WRK_throttle,10 - (1 - (WRK_TemperatureSetpoint - ActualTemperature) / 40) * 10) ,GEQ(ActualTemperature,WRK_TemperatureSetpoint) CLR(WRK_throttle) ,CMP(WRK_TemperatureSetpoint - ActualTemperature > 40) MOV(10,WRK_throttle) ];
   // Temperature "Simulation"
   // Lines 328-336, 347-366 of C#  [ UpdateOvenTemperature() ]
   2: NEQ(ActualTemperature,WRK_TemperatureSetpoint)CPT(ActualTemperature,ActualTemperature + (WRK_TemperatureSetpoint - ActualTemperature) * 0.1);
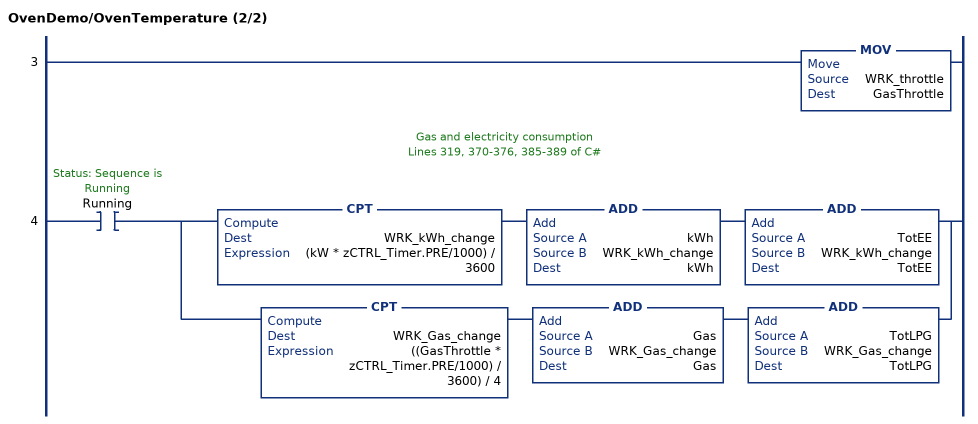
   3: MOV(WRK_throttle,GasThrottle);
   // Gas and electricity consumption
   // Lines 319, 370-376, 385-389 of C#
   4: XIC(Running)[CPT(WRK_kWh_change,(kW * zCTRL_Timer.PRE/1000) / 3600) ADD(kWh,WRK_kWh_change,kWh) ADD(TotEE,WRK_kWh_change,TotEE) ,CPT(WRK_Gas_change,((GasThrottle * zCTRL_Timer.PRE/1000) / 3600) / 4) ADD(Gas,WRK_Gas_change,Gas) ADD(TotLPG,WRK_Gas_change,TotLPG) ];
END_ROUTINE
END_PROGRAM
